// TIA Portal project "Project1" (V12)

(* hardware
DEVICE "S7-1200 station_1"  SIMATIC 1200-Station
   slot 0: "S7-1200 rack"  Rack  V1.0
   slot 1: "PLC_1"  CPU 1214C DC/DC/DC  6ES7 214-1AG31-0XB0  V3.0
*)

// ===== PLC "PLC_1"  CPU 1214C DC/DC/DC =====

VAR_GLOBAL   // PLC tag table "Default tag table"
   "Tag_1" AT %I0.0 : Bool;
   "Tag_2" AT %Q0.0 : Bool;
   "Tag_3" AT %M0.4 : Bool;
   "Tag_4" AT %M0.1 : Bool;
   "Tag_5" AT %M1.0 : Bool;
   "Tag_6" AT %M1.3 : Bool;
   "Tag_7" AT %IW64 : Word;
   "Tag_8" AT %MW10 : Word;
   "Tag_9" AT %MD12 : Real;
   "Tag_10" AT %MD16 : Real;
   "Tag_11" AT %MW12 : Word;
   "Tag_12" AT %MW16 : Word;
   "Tag_13" AT %MW20 : UInt;
   "Tag_14" AT %MW24 : UInt;
END_VAR

ORGANIZATION_BLOCK "Main"   // OB1, LAD, ProgramCycle
TITLE = "Main Program Sweep (Cycle)"
{ S7_Optimized_Access := 'FALSE' }
VERSION : 0.1
BEGIN

REGION Network 1
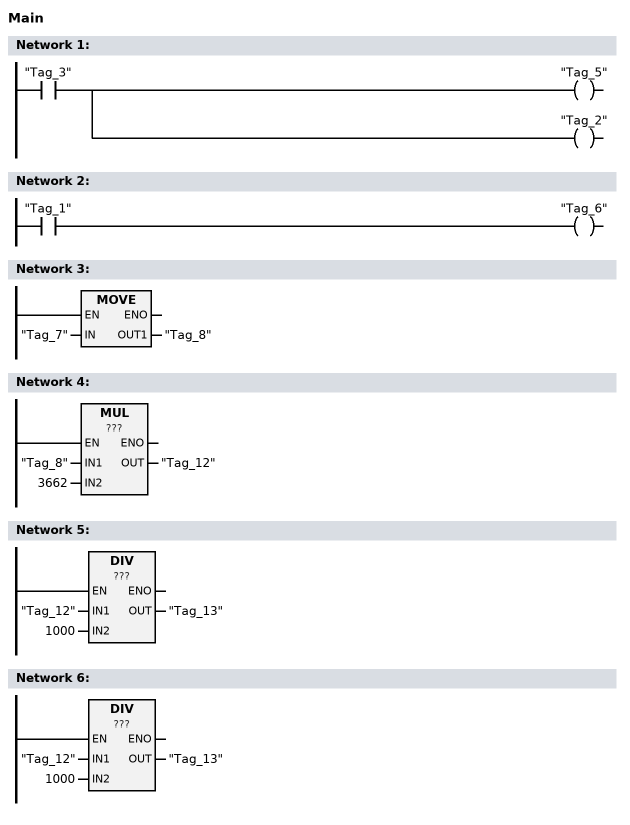
   RUNG wire#powerrail
      Contact( "Tag_3" )
      wire#w1
      Coil( "Tag_5" )
   END_RUNG
   RUNG wire#w1
      Coil( "Tag_2" )
   END_RUNG
   // the same network as SCL:
   "Tag_5" := "Tag_3";
   "Tag_2" := "Tag_3";
END_REGION

REGION Network 2
   RUNG wire#powerrail
      Contact( "Tag_1" )
      Coil( "Tag_6" )
   END_RUNG
   // the same network as SCL:
   "Tag_6" := "Tag_1";
END_REGION

REGION Network 3
   RUNG wire#powerrail
      { S7_GenerateENO := "TRUE" } Move(in := "Tag_7", out1 => "Tag_8")
   END_RUNG
   // the same network as SCL:
   "Tag_8" := "Tag_7";
END_REGION

REGION Network 4
   RUNG wire#powerrail
      { S7_Templates := "SrcType := ???"; S7_GenerateENO := "TRUE" } Mul(in1 := "Tag_8", in2 := 3662, out => "Tag_12")
   END_RUNG
   // the same network as SCL:
   "Tag_12" := "Tag_8" * 3662;
END_REGION

REGION Network 5
   RUNG wire#powerrail
      { S7_Templates := "SrcType := ???"; S7_GenerateENO := "TRUE" } Div(in1 := "Tag_12", in2 := 1000, out => "Tag_13")
   END_RUNG
   // the same network as SCL:
   "Tag_13" := "Tag_12" / 1000;
END_REGION

REGION Network 6
   RUNG wire#powerrail
      { S7_Templates := "SrcType := ???"; S7_GenerateENO := "TRUE" } Div(in1 := "Tag_12", in2 := 1000, out => "Tag_13")
   END_RUNG
   // the same network as SCL:
   "Tag_13" := "Tag_12" / 1000;
END_REGION
END_ORGANIZATION_BLOCK